ACTION _CalData:
// nOutputMode
// 0 : uses setpoint and setpoint type to control the valve.
// 1 : Does not use setpoint and setpoint type to operate the valve.
// 2 : Does not use setpoint and setpoint type to operate the valve.
// 3 : Holds valve in current position.
// 4 : Reset the controller.

GVL_IO.nIQPLUS_SetType 	:= GVL_DEVICE_NET_IQ_PLUS.nOutputSetType;
GVL_IO.nIQPLUS_Mode 	:= GVL_DEVICE_NET_IQ_PLUS.nOutputMode;
GVL_DEVICE_NET_IQ_PLUS.nOutputMode := GVL_COMMAND_FROM_UI.CMD_THROTTLE_OUTPUT_MODE;
GVL_IO.aMonitoring_PV[E_Morning_Index.E_Morning_TV_Position] := wByteValvePosition_PV/SetPointFactor;

(* Read from Device Value *)
// 2USINT to WORD
wByteCDG1_PV 		:= USINT_TO_WORD_jh(GVL_DEVICE_NET_IQ_PLUS.aInputPressurePV_CDG1);
wByteCDG2_PV 		:= USINT_TO_WORD_jh(GVL_DEVICE_NET_IQ_PLUS.aInputPressurePV_CDG2);
wByteValvePosition_PV:= USINT_TO_WORD_jh(GVL_DEVICE_NET_IQ_PLUS.aInputValvePosionPV);
wByteValvePosition_PV_Monitoring:=REAL_TO_WORD(wByteValvePosition_PV/SetPointFactor);
GVL_IO.aMonitoring_PV[12] := wByteValvePosition_PV_Monitoring;




wControlValue		:= GVL_IO.wIqPlus_CV;

//From IQ Plus
CDG1_RealValue :=wByteCDG1_PV/PressureFactor; 
GVL_IO.wIqPlus_CDG1_PV 	:= REAL_TO_WORD(wByteCDG1_PV/PressureFactor);
GVL_IO.wIqPlus_CDG2_PV:=GVL_IO.wIqPlus_CDG1_PV;

IF GVL_IO.wIqPlus_CDG1_PV > 800 OR GVL_IO.wIqPlus_CDG1_PV <=1 THEN
	GVL_IO.wIqPlus_CDG1_PV:=0;
	GVL_IO.wIqPlus_CDG2_PV:=0;
END_IF

CDG_1_Value_RealType:=wByteCDG1_PV/PressureFactor;


//nSetType //1:Pressure Conrol, 2:Position Control

IF GVL_DEVICE_NET_IQ_PLUS.nOutputMode = 0 AND nSetType = 1 THEN(*Pressure Mode*)
	wTypedControlValue := REAL_TO_WORD(wControlValue * SetPointFactor * 0.1); //Pressure Control
ELSIF GVL_DEVICE_NET_IQ_PLUS.nOutputMode = 0 AND nSetType = 2 THEN (*Position Mode*)
	wTypedControlValue := REAL_TO_WORD(wControlValue * SetPointFactor); // Position Control
END_IF

wOutputSVBytes 		:= WORD_TO_USINT_Bit(wTypedControlValue);
GVL_DEVICE_NET_IQ_PLUS.aOutputSVBytes[1] 	:= wOutputSVBytes.Lower;
GVL_DEVICE_NET_IQ_PLUS.aOutputSVBytes[2] 	:= wOutputSVBytes.Upper;

//Valve Status Initailize
IF GVL_DEVICE_NET_IQ_PLUS.nInputStatus <> nInputStatusOld THEN
	// Staus Initializing
	ingPressureControl := FALSE;
	ingPositionControl := FALSE;
	isValveOpen := FALSE;
	isValveNotInitialized := FALSE;	
	isValveClosed := FALSE;
	isValveFaultState := FALSE;
	ingValveInitializing := FALSE;
	ingHoldState := FALSE;
	isPressureControl:=FALSE;
	// Status Update	
	nInputStatusOld := GVL_DEVICE_NET_IQ_PLUS.nInputStatus;
END_IF

//Update Valve Status
CASE GVL_DEVICE_NET_IQ_PLUS.nInputStatus OF
	0 : ingPressureControl := TRUE; //Pressure Control Performing.
	1 : ingPositionControl := TRUE; //Position Control Performing.	
	2 : isValveOpen := TRUE; //Valve Open, Stopped, Not Controlling.
	3 : isValveNotInitialized := TRUE; //Valve not initialized power on or RESET Command.
	4 : isValveClosed := TRUE; //Valve Closed, Stopped, Not Controlling.
	5 : isValveFaultState := TRUE; //Has faulted during valve initialization or operation.
	6 : ingValveInitializing := TRUE; //Initailizing Process.
	7 :	isPressureControl:=TRUE;
	8 : ingHoldState := TRUE; //intermediate position, not at open or close and not controlling pressure.
END_CASE
END_ACTION

ACTION _DigitalInput:

(* Command *)

bPumpOn:= GVL_COMMAND_FROM_UI.CMD_VACUUM_PUMP_ON;
bPumpReset:=GVL_COMMAND_FROM_UI.CMD_VACUUM_PUMP_RESET;
(* Read from Power Distribution Pannel *)
bVacuumPumpCB		:= GVL_IO_GAS_CABINET.DI_02_VacuumPumpELCB;
bThrottleValveCP 	:= GVL_IO_GAS_CABINET.DI_02_T_VCP;

(* Read from Vacuum Pump *)
isPumpFault			:= GVL_IO_REACTOR_CABINET.DI_02_VacuumPumpFail;
isPumpWarning		:= GVL_IO_REACTOR_CABINET.DI_02_VacuumPumpWarning;
isPumpAlarm			:= GVL_IO_REACTOR_CABINET.DI_02_VacuumPumpAlarm;
isPumpRunning		:= GVL_IO_REACTOR_CABINET.DI_02_VacuumPumpFBRunning;
isFBRunning			:= GVL_IO_REACTOR_CABINET.DI_02_VacuumPumpRunning;


GVL_IO.isPumpRunning := GVL_IO_REACTOR_CABINET.DI_02_VacuumPumpFBRunning;
END_ACTION

ACTION _DigitalOutput:
//GVL_IO.aDigitalOutputIO[2].2 := bPumpOn; //Pump On
//GVL_IO.aDigitalOutputIO[2].3 := bPumpReset; // Pump Reset

GVL_IO_REACTOR_CABINET.DO_05_VacuumPumpStart_Stop := bPumpOn;
GVL_IO_REACTOR_CABINET.DO_05_VacuumPumpReset := bPumpReset;
END_ACTION

END_PROGRAM

// ---- POUs/P13_LineHeater.TcPOU
PROGRAM P13_LineHeater
VAR
	rTemperatureSV 		: ARRAY[1..8]OF REAL;
	bAutoTuneSV 		: ARRAY[1..8]OF BOOL;

	rTemperaturePV 		: ARRAY[1..8]OF REAL;
	isLineHeater_Run	: ARRAY[1..8]OF BOOL;
	isLineHeater_ATune	: ARRAY[1..8]OF BOOL;
	isLineHeater_Err	: ARRAY[1..8]OF BOOL;

	TimeOnDelay			: TON; //Time delay after Power ON of Thermal Bath
	TimeCycle			: TON;
	nComMode 			: INT; // //1 = PV Req, 2 = STATUS Req, 3 = SV Write, 4 = AutoTune On/Off
	nCount 				: INT;
	rTemperatureTV 		: ARRAY[1..8]OF REAL;
	bAutoTuneTV			: ARRAY[1..8]OF BOOL;

	//for sending variable
	TimeWaitSend		:TON;
	bSendingEnable 		: BOOL:=TRUE; // Check the Sending Stage
	bSetValueMode 		: BOOL;
	fbSend				: SendString;
	sSendString 		: STRING;
	bSendBusy			: BOOL;
	bSendingOK 			: BOOL; //v1
	eSendErrorID		: ComError_t;
	
	// for received variable
	TimeWaitReceive		:TON;
	fbReceive			: ReceiveString;
	sReceivedString		: STRING;
	bStringReceived		: BOOL;
	bReceiveBusy		: BOOL;
	bReceiveError		: BOOL;
	eReceiveErrorID		: ComError_t;
	bReceiveTimeout		: BOOL;
	bReceivedOK 		: BOOL;
	hStrReceivedST		: STRING;
	hStrReceivedPV		: STRING;
	
	nHeaterNumber 		: INT := 1;
	sHeaterNumber 		: STRING := '1';
	sReceivedHeaterNumber : STRING;
	nReceivedHeaterNumber : INT;
	sReceivedAffirmation : STRING;
	sReceivedData 		: STRING;
	nHeaterStrPositionPV : INT:= 11; //Received String Start Position
	nDecimal			:INT;
	nSendStrCounter		:INT := 1;
	bReset : BOOL;
	sTest : STRING;
	nStrPosition : INT;
	nHeaterNumberPV : INT;
	sTemperaturePV : STRING;
	(* Input *)
	bLineHeaterCB		: BOOL;
	bLineHeaterCP		: BYTE;
END_VAR

_DIgitalInput();

TimeOnDelay(IN:= GVL_IO_GAS_CABINET.DI_02_LineHeatersELCB, PT :=T#5S); //Time Delay after a Thermal Bath MC ON

IF TimeOnDelay.Q THEN
	TimeOnDelay(IN:=FALSE);
	FOR nHeaterNumber:= 1 TO 8 DO
		IF (rTemperatureTV[nHeaterNumber] <> rTemperatureSV[nHeaterNumber]) THEN
			// if SetValue are different to TargetValue, change Target vale to setvalue
			rTemperatureTV[nHeaterNumber] := rTemperatureSV[nHeaterNumber];
			
			_SendTemp();
		END_IF
	END_FOR
END_IF


rTemperaturePV[1] := GVL_Serial.LineHeater_data_1.LINE_HEATER_CH_1_PV_VALUE;
rTemperaturePV[2] := GVL_Serial.LineHeater_data_1.LINE_HEATER_CH_2_PV_VALUE;
rTemperaturePV[3] := GVL_Serial.LineHeater_data_1.LINE_HEATER_CH_3_PV_VALUE;
rTemperaturePV[4] := GVL_Serial.LineHeater_data_1.LINE_HEATER_CH_4_PV_VALUE;

rTemperaturePV[5] := GVL_Serial.LineHeater_data_2.LINE_HEATER_CH_1_PV_VALUE;
rTemperaturePV[6] := GVL_Serial.LineHeater_data_2.LINE_HEATER_CH_2_PV_VALUE;
rTemperaturePV[7] := GVL_Serial.LineHeater_data_2.LINE_HEATER_CH_3_PV_VALUE;
rTemperaturePV[8] := GVL_Serial.LineHeater_data_2.LINE_HEATER_CH_4_PV_VALUE;

GVL_IO.aLineHeater_rTemperaturePV := rTemperaturePV;

ACTION _DigitalInput:
bLineHeaterCB	:= GVL_IO_GAS_CABINET.DI_02_LineHeatersELCB;

bLineHeaterCP.0 	:= GVL_IO_GAS_CABINET.DI_03_LineHeater_1CP;
bLineHeaterCP.1 	:= GVL_IO_GAS_CABINET.DI_03_LineHeater_2CP;
bLineHeaterCP.2 	:= GVL_IO_GAS_CABINET.DI_03_LineHeater_3CP;
bLineHeaterCP.3 	:= GVL_IO_GAS_CABINET.DI_03_LineHeater_4CP;
bLineHeaterCP.4 	:= GVL_IO_GAS_CABINET.DI_03_LineHeater_5CP;
bLineHeaterCP.5 	:= GVL_IO_GAS_CABINET.DI_04_LineHeater_6CP;
bLineHeaterCP.6 	:= GVL_IO_GAS_CABINET.DI_04_LineHeater_7CP;
bLineHeaterCP.7 	:= GVL_IO_GAS_CABINET.DI_04_LineHeater_8CP;
END_ACTION

ACTION _SendTemp:
CASE nHeaterNumber OF
	1:
		GVL.fbLineHeater_Manager._SendModbusCommand(sendMessage:=F_Temp_Write_Set_Point(Module_Number:=1,CommandIndex:=16#0
																,Write_Value:=REAL_TO_WORD(rTemperatureSV[nHeaterNumber])));
	2:
		GVL.fbLineHeater_Manager._SendModbusCommand(sendMessage:=F_Temp_Write_Set_Point(Module_Number:=1,CommandIndex:=16#03E8
																,Write_Value:=REAL_TO_WORD(rTemperatureSV[nHeaterNumber])));
	3:
		GVL.fbLineHeater_Manager._SendModbusCommand(sendMessage:=F_Temp_Write_Set_Point(Module_Number:=1,CommandIndex:=16#07D0
																,Write_Value:=REAL_TO_WORD(rTemperatureSV[nHeaterNumber])));
	4:
		GVL.fbLineHeater_Manager._SendModbusCommand(sendMessage:=F_Temp_Write_Set_Point(Module_Number:=1,CommandIndex:=16#0BB8
																,Write_Value:=REAL_TO_WORD(rTemperatureSV[nHeaterNumber])));
																
	(*Change Module Number*)															
	5:
		GVL.fbLineHeater_Manager._SendModbusCommand(sendMessage:=F_Temp_Write_Set_Point(Module_Number:=2,CommandIndex:=16#0
																,Write_Value:=REAL_TO_WORD(rTemperatureSV[nHeaterNumber])));
	6:
		GVL.fbLineHeater_Manager._SendModbusCommand(sendMessage:=F_Temp_Write_Set_Point(Module_Number:=2,CommandIndex:=16#03E8
																,Write_Value:=REAL_TO_WORD(rTemperatureSV[nHeaterNumber])));
	7:
		GVL.fbLineHeater_Manager._SendModbusCommand(sendMessage:=F_Temp_Write_Set_Point(Module_Number:=2,CommandIndex:=16#07D0
																,Write_Value:=REAL_TO_WORD(rTemperatureSV[nHeaterNumber])));
	8:
		GVL.fbLineHeater_Manager._SendModbusCommand(sendMessage:=F_Temp_Write_Set_Point(Module_Number:=2,CommandIndex:=16#0BB8
																,Write_Value:=REAL_TO_WORD(rTemperatureSV[nHeaterNumber])));
END_CASE
END_ACTION

END_PROGRAM

// ---- POUs/P14_ThermalBath.TcPOU
PROGRAM P14_ThermalBath
VAR
	rTemperatureSV 		: ARRAY[1..6]OF REAL;

	(* Input from Device *)
	bTempDeviationAlarm	: ARRAY[1..6] OF BOOL;
	bCutOffAlarm		: ARRAY[1..6] OF BOOL;
	
	rTemperature_PV 		: ARRAY[1..6]OF REAL;
	isBath_Err 			: ARRAY[1..6]OF BOOL;
	isBath_TC_Broken 	: ARRAY[1..6]OF BOOL ; 

	//for send variable
	TimeOnDelay	: TON; //Time delay after Power ON of Thermal Bath
	TimeCycle			: TON;
	TimeWaitSend		: TON;
	TimeWaitReceive		: TON;
	bSendingEnable 		: BOOL:=TRUE; // Check the Sending Stage
	bSetValueMode 		: BOOL;
	rTemperatureTV 		: ARRAY[1..6]OF REAL;
	fbSend				: SendString;
	sSendString 		: STRING;
	bSendBusy			: BOOL;
	bSendingOK 			: BOOL;
	eSendErrorID		: ComError_t;

	// for received variable
	fbReceive			: ReceiveString;
	sReceivedString		: STRING;
	bStringReceived		: BOOL;
	bReceiveBusy		: BOOL;
	bReceiveError		: BOOL;
	eReceiveErrorID		: ComError_t;
	bReceiveTimeout		: BOOL;
	bReceivedOK 		: BOOL;
	
	nBathNumber 		: INT := 1;
	sBathNumber 		: STRING := '1';
	sReceivedBathNumber : STRING;
	nReceivedBathNumber : INT;
	sReceivedAffirmation : STRING;
	sReceivedData 		: STRING;
	
	(* Input *)
	bThermalBathCB		: BOOL;
	index				: INT;
END_VAR

// Call the send block every second to repeat the transmission.
// Also call the block as long as it is busy to finish a transmission.
//TB: Thermal Bath x 6EA
//Maker: SMC
//Model: HEBC002-WA10
//Temp Range: -15 ~60℃
//RS485: 9600, DataBit(8), Parity(None), StopBit(1)
//BCC Check X

(* Read from Power Distribution Pannel *)
_DigitalInput();

// make a sending string
TimeCycle(IN := TimeOnDelay.Q, PT := T#1S); //Cycle for Serial Communication
IF TimeCycle.Q = TRUE THEN
	TimeCycle(IN := FALSE);

	// Make a sending string Set value or Request value 
	IF bSendingEnable = TRUE THEN
		//Set sate
		bSendingEnable := FALSE;
		bReceivedOK := FALSE;
		bSetValueMode := FALSE;
		
		//Target value(Bath) Set value
		IF (rTemperatureTV[nBathNumber] <> rTemperatureSV[nBathNumber])  OR isBath_Err[nBathNumber] THEN
			
			rTemperatureTV[nBathNumber] := rTemperatureSV[nBathNumber];
			
			sSendString := Real_To_String_ThermalBath(rTemperatureTV[nBathNumber],nBathNumber); //Send a SetValue=10.0 '$0201WSV100100$03'
			bSetValueMode := TRUE;
		ELSE
			sBathNumber := INT_TO_STRING(nBathNumber);
			sSendString := INSERT('$020RPV1$03',sBathNumber,2); //Request a PV
			bSetValueMode := FALSE;
		END_IF
		
		// Send string	
		fbSend(	SendString:= sSendString,
			TXbuffer:= GVL_Serial.TxBufferTB,
			
			Busy=> bSendBusy,
			Error=> );
		IF fbSend.Error <> COMERROR_NOERROR THEN
			eSendErrorID := fbSend.Error;
			bSendingOK := FALSE;
		ELSE
			eSendErrorID := COMERROR_NOERROR;
			bSendingOK := TRUE;
		END_IF
		
	END_IF

	//	Receive string data:
	//	The block receives any data strings beginning with a STX ($02) and ending with an ETX ($03) character.
	TimeWaitReceive(IN := bSendingOK, PT := T#250MS); //Wait receiving data
	IF TimeWaitReceive.Q THEN
		TimeWaitReceive(IN:= FALSE);
		fbReceive(
			Prefix:= '$02',
			Suffix:= '$03',
			Timeout:= T#1S,
			ReceivedString:= sReceivedString,
			RXbuffer:= GVL_Serial.RxBufferTB,
			
			StringReceived=> bStringReceived,
			Busy=> bReceiveBusy,
			Error=> ,
			RxTimeout=> bReceiveTimeout );
			
		IF bReceiveTimeout THEN
			isBath_Err[nReceivedBathNumber] := TRUE;
			bReceiveTimeout := FALSE;
		END_IF
		
		IF fbReceive.Error <> COMERROR_NOERROR THEN
			eReceiveErrorID := fbReceive.Error;
		END_IF
		
		IF bStringReceived THEN
			bStringReceived :=FALSE;
			bReceivedOK := TRUE;
			bSendingEnable := TRUE;
			sReceivedBathNumber := MID(STR:=sReceivedString, len:=1, pos:=3); //ReceivedString : '$0201$06PV100250$03'
			nReceivedBathNumber := STRING_TO_INT(sReceivedBathNumber);
			sReceivedAffirmation := MID(STR:=sReceivedString, len:=1, pos:=4); //Affirmation
			
			IF bSetValueMode THEN //Write SV Mode
				IF sReceivedAffirmation = '$06' THEN //'$06' ReceivedString : '$0201$06$03'
					isBath_Err[nReceivedBathNumber] := FALSE;
				ELSE
					//isBath_Err[nReceivedBathNumber] := TRUE;
				END_IF
				bSetValueMode := FALSE;
			ELSE //Read PV Mode
				sReceivedData := MID(STR:=sReceivedString, len:=5, pos:=8); //ReceivedString : '$0201$06PV100250$03'
				IF sReceivedData = '' THEN
					//isBath_Err[nReceivedBathNumber] := TRUE;
				ELSIF sReceivedData = 'HHHHH' THEN
					rTemperature_PV[nReceivedBathNumber] := -99.0;
					isBath_TC_Broken[nReceivedBathNumber] := TRUE;
					isBath_Err[nReceivedBathNumber] := FALSE;
				ELSE
					rTemperature_PV[nReceivedBathNumber] := (STRING_TO_REAL(sReceivedData))/10;
					isBath_TC_Broken[nReceivedBathNumber] := FALSE;
					isBath_Err[nReceivedBathNumber] := FALSE;
				END_IF
			END_IF
			index := nReceivedBathNumber + 11;
			
			
		END_IF
	END_IF
	
	//Change the Next Bath
	nBathNumber := nBathNumber + 1;
	IF nBathNumber > 4 THEN
		nBathNumber := 1;
	END_IF
	bSendingEnable := TRUE;
END_IF

ACTION _DigitalInput:
//bThermalBathCB := GVL_IO.aDigitalInputIO[5].0;
bThermalBathCB := GVL_IO_GAS_CABINET.DI_02_ThermalBathsELCB;

(* Read from SMC Bath Device Value *)
//TimeOnDelay(IN:= P90_Interlock.bThermalBathMC, PT :=T#1S); //Time Delay after a Thermal Bath MC ON
TimeOnDelay(IN:= GVL_IO_GAS_CABINET.DI_02_ThermalBathsELCB, PT :=T#1S); //Time Delay after a Thermal Bath MC ON

bTempDeviationAlarm[1]	:= GVL_IO_GAS_CABINET.DI_05_ThermalBath_1DeviationAlarm;
bTempDeviationAlarm[2]	:= GVL_IO_GAS_CABINET.DI_05_ThermalBath_2DeviationAlarm;
bTempDeviationAlarm[3]	:= GVL_IO_GAS_CABINET.DI_06_ThermalBath_3DeviationAlarm;
bTempDeviationAlarm[4]	:= GVL_IO_GAS_CABINET.DI_06_ThermalBath_4DeviationAlarm;

bCutOffAlarm[1] := NOT(GVL_IO_GAS_CABINET.DI_05_ThermalBath_1CutOffAlarm); //Normally Contact
bCutOffAlarm[2] := NOT(GVL_IO_GAS_CABINET.DI_05_ThermalBath_2CutOffAlarm); 
bCutOffAlarm[3] := NOT(GVL_IO_GAS_CABINET.DI_06_ThermalBath_3CutOffAlarm); 
bCutOffAlarm[4] := NOT(GVL_IO_GAS_CABINET.DI_06_ThermalBath_4CutOffAlarm);
END_ACTION

END_PROGRAM

// ---- POUs/P15_RotationOperation.TcPOU
PROGRAM P15_RotationOperation
VAR
	rControlValue			: REAL; //rpm
	bStart_Stop				: BOOL := TRUE;
	bAlarmReset				: BOOL; //Motor Driver Alarm

	bRotationCP				: BOOL;
	nConvertedRotation_PV	: REAL; //PV 0~100 rpm

	rConvertedCV			:REAL;
	(* Motor Driver *)
	bBrake_Run				: BOOL;
	(* Rotation Operation Parameter*)
	wRotaion_PV				: WORD;
	isRotationFault			: BOOL; //Motor Driver
	calcRotation: REAL;
END_VAR

VAR CONSTANT
	KL4404MaxValueP		: REAL := 16383; //0~5V, 0~3000
	//Motor Max Rotation RPM 3000rpm, Gear Ratio 20, Belt Ratio 4.5
	ConversionFactor 	: REAL :=491.49;// 491.49 ; //13106 * 20 * 4.5 / 3000
END_VAR

// Oriental Motor Driver : BLHM230K-GFS, 0~4V

_DigitalInput();

calcRotation := (wRotaion_PV / ConversionFactor) * (5.0/3.0);


nConvertedRotation_PV := (calcRotation);

// Interface with other PRGs
GVL_IO.nRotation_Converted_PV := nConvertedRotation_PV;
rControlValue := GVL_IO.rRotation_ControlValue;

//Write to Motor Driver
rConvertedCV := rControlValue * ConversionFactor; // Convert from RPM to control value


IF GVL_io.aInterlockEnable[1].7 = TRUE THEN // UI 의 Auto Power ON 기능에 따라서 자동 On . oFF 사용 
	IF (GVL_IO.aController[E_aAnalogInputIO_Index.E_PV_susceptorRotation].input.targetValue > 0) OR (rConvertedCV > 0) THEN // Motor Driver RUN
		bBrake_Run := TRUE;
	ELSIF (GVL_IO.aController[E_aAnalogInputIO_Index.E_PV_susceptorRotation].input.targetValue = 0) AND (rConvertedCV = 0) THEN
		bBrake_Run := FALSE;
	END_IF
ELSE
	bBrake_Run:=FALSE;
END_IF

_DigitalOutput();

ACTION _DigitalInput:
(* Read from Power Distribution Pannel *)
bRotationCP := GVL_IO_GAS_CABINET.DI_02_RotationMotorCP;

//from Device Value
isRotationFault := NOT(GVL_IO_REACTOR_CABINET.DI_02_SusceptorRotationMotorFault);
wRotaion_PV := INT_TO_WORD(GVL_IO_REACTOR_CABINET.AI_08_R01SusceptorRotationPV);
END_ACTION

ACTION _DigitalOutput:
GVL_IO_REACTOR_CABINET.DO_05_SusceptorRotationFWD := bBrake_Run;
GVL_IO_REACTOR_CABINET.AO_09_R01_SusceptorRotationSV:=REAL_TO_INT(rConvertedCV);
END_ACTION

END_PROGRAM

// ---- POUs/P16_CoverOperation.TcPOU
PROGRAM P16_CoverOperation
VAR
// 	isCoverClosed 	: BOOL;

	bCoverCP	: BOOL;
	bLowerLimit	: BOOL;
	bUpperLimit	: BOOL;
	TimerUpLED 		: TON;
	TimerUpLED_X 	: TON;
	TimerDownLED 	: TON;
	TimerDownLED_X 	: TON;
	TimerDownDelayOff 	: TON;
	(* Input *)
	bUpSwitch	: BOOL;
	bDownSwitch 	: BOOL;
	bClamp_Lock_switch: BOOL;
	bClamp_Release_switch: BOOL;
	(* Output *)
	bUpLED 		: BOOL;
	bDownLED 	: BOOL;
	bOnUpRelay 	: BOOL;
	bOnDownRelay : BOOL;
	bOnClamp_Lock_Relay:BOOL;
	bOnClamp_Release_Relay:BOOL;		
	
	bClampLock: BOOL;
	bClampRelease: BOOL;
END_VAR

_DigitalInput();

TimerDownDelayOff(IN:=bLowerLimit, PT:=T#500MS);

//Cover Open 조건
//공정 중이지 않을것
//Dor Pressure down
//Clamp Releaae
//Susceptor down
//CDG 700 torr 이상
//모든 벨브 ff

// Cover Operation Condition
IF P90_Interlock.bReactorOpenEnable THEN
	(*Cover*)
	IF bClampRelease THEN
		bOnUpRelay := (bDownSwitch = FALSE AND bUpSwitch = TRUE AND bUpperLimit = FALSE );
		bOnDownRelay := (bDownSwitch = TRUE AND bUpSwitch = FALSE AND (bLowerLimit = FALSE OR TimerDownDelayOff.Q = FALSE ));
	ELSE
		bOnUpRelay:=FALSE;
		bOnDownRelay:=FALSE;
	END_IF
	(*clamp*)
	bOnClamp_Lock_Relay:=(bClamp_Lock_switch = TRUE AND bClamp_Release_switch = FALSE);
	bOnClamp_Release_Relay:=(bClamp_Lock_switch = FALSE AND bClamp_Release_switch = TRUE);
ELSE
	(*Cover*)
	bOnUpRelay:=FALSE;
	bOnDownRelay:=FALSE;
	(*clamp*)
	bOnClamp_Lock_Relay:=FALSE;
	bOnClamp_Release_Relay:=FALSE;
END_IF

//LED Blinking
TimerUpLED(IN:=(bOnUpRelay AND TimerUpLED_X.Q = FALSE), PT:=T#500MS);
TimerUpLED_X(IN:=TimerUpLED.Q, PT:=T#300MS);
bUpLED := (TimerUpLED.Q AND bOnUpRelay) OR bUpperLimit;

TimerDownLED(IN:=(bOnDownRelay AND TimerDownLED_X.Q = FALSE), PT:=T#500MS);
TimerDownLED_X(IN:=TimerDownLED.Q, PT:=T#300MS);
bDownLED := (TimerDownLED.Q AND bOnDownRelay) OR bLowerLimit;

_DigitalOutput();

ACTION _DigitalInput:
//(* Read from Device Value *)
//// Cover Operation Switch
//bUpSwitch 		:= GVL_IO.aDigitalInputIO[1].6;
//bDownSwitch 	:= GVL_IO.aDigitalInputIO[1].7;
//bUpperLimit 	:= GVL_IO.aDigitalInputIO[3].4;
//bLowerLimit 	:= GVL_IO.aDigitalInputIO[3].5;
//bCoverCP 		:=  GVL_IO.aDigitalInputIO[5].4;

bUpSwitch 		:=GVL_IO_REACTOR_CABINET.DI_01_ReactorDoorUpButton;
bDownSwitch 	:=GVL_IO_REACTOR_CABINET.DI_01_ReactorDoorDownButton;
bUpperLimit 	:=GVL_IO_REACTOR_CABINET.DI_02_ReactorDoorUpLimitSensor;
bLowerLimit 	:=GVL_IO_REACTOR_CABINET.DI_03_ReactorDoorDownLimitSensor;
bCoverCP 		:= GVL_IO_GAS_CABINET.DI_02_CoverLiftMotorCP;

bClampLock := GVL_IO_REACTOR_CABINET.DI_03_CylinderAutoSwitch_Closed;
bClampRelease :=GVL_IO_REACTOR_CABINET.DI_03_CylinderAutoSwitch_Opened;

bClamp_Lock_switch:=GVL_IO_REACTOR_CABINET.DI_01_ClampLock;
bClamp_Release_switch:=GVL_IO_REACTOR_CABINET.DI_01_ClampRelease;
END_ACTION

ACTION _DigitalOutput:
(* Write to Device Value *)
// Cover Operation Switch Lamp


//Status Output
GVL_IO.isCoverClosed := bLowerLimit;

GVL_IO_REACTOR_CABINET.DO_06_ReactorCoverUpButtonLamp := bUpLED;
GVL_IO_REACTOR_CABINET.DO_06_ReactorCoverDownButtonLamp := bDownLED;

GVL_IO_REACTOR_CABINET.DO_04_ReactorCoverUpRelay :=bOnUpRelay;
GVL_IO_REACTOR_CABINET.DO_04_ReactorCoverDownRelay :=bOnDownRelay;

GVL_IO_REACTOR_CABINET.DO_06_ClampLockButtonLamp := GVL_IO_REACTOR_CABINET.DI_03_CylinderAutoSwitch_Closed;
GVL_IO_REACTOR_CABINET.DO_06_ClampReleaseButtonLamp := GVL_IO_REACTOR_CABINET.DI_03_CylinderAutoSwitch_Opened;

GVL_IO_REACTOR_CABINET.DO_05_ClampLock := bOnClamp_Lock_Relay;
GVL_IO_REACTOR_CABINET.DO_05_ClampRelease := bOnClamp_Release_Relay;
END_ACTION

END_PROGRAM

// ---- POUs/P17_DOROperation.TcPOU
PROGRAM P17_DOROperation
VAR
	bDOROn				: BOOL; //UI Input Button
	bDOROff				: BOOL; //UI Input Button
	fTresholdPressure	: REAL;
	fTresholdCount		: REAL;
	bPressureEnable 	: BOOL;
	bCountEnable		: BOOL;

	isDOROnState		: BOOL := FALSE; //DOR ON State
	bError				: INT; //0: No Err, 1: Vacuum Fail, 2: Vacuum Release, 3: Try out
	nWaitCounter		: INT;

	(* Input *)
	bVacSwitch			: BOOL; //Push Switch
	bAtmSwitch			: BOOL; //Push Switch
	(* Pressure Transducer *)
	nPressurePV			: INT;
	rPressurePV_kPa		: REAL;
	(* Output *)
	bVacLED				: BOOL;
	bAtmLED				: BOOL;
	bV_DORVac			: BOOL; //V34 Valve
	bV_DORFill			: BOOL; //V35 Valve
	
	(* DOR Condition Operation Parameter *)
	rTrigSwitch			: R_TRIG;
	TimerOnLED			: TON;
	TimerVacSwitch		: TON;
	TimerAtmSwitch		: TON;
	TimerWaitCheck		: TON;
	TimerVacRealease	: TON;
	nCase				: INT := 0;
	nTresholdCount		: INT;
	nTryCount			: INT;
	bVacuumRealse		: BOOL;
	//Temperatur Variable
	bTest				: BOOL;
	nTest				: INT;
END_VAR

VAR CONSTANT
	KL3464MaxValueP		: REAL := 16383; //1 ~ 5VDC, 0 ~ 100kPa(1bar), PG35
	SlopeFactor			: REAL := 0.007617887; //100kPa/(16383-3256)
END_VAR

// Double O-Ring Vacuum Condition

_DigitalInput();

(* If Vacuum 'ON' Switch Press, Change DOR Vacuum State *)
//DOR Operation Signal generation

TimerVacSwitch(IN:=bVacSwitch OR bDOROn, PT:=T#100MS);
rTrigSwitch(CLK:=TimerVacSwitch.Q);

IF rTrigSwitch.Q AND GVL_IO.bDorOnEnable THEN
	nCase 		:= 1;
	nTryCount 	:= 1; //Try One more Vacuum 
END_IF

CASE nCase OF
	1: //Initialize
		isDOROnState := FALSE;
		bV_DORVac 	:= TRUE; //V34 Open
		bV_DORFill	:= FALSE; //V35 Close
		bAtmLED		:= FALSE;
		TimerWaitCheck(IN:=FALSE);	
		nCase := 10;
	10: //Wait and Vacuum Check
		(* Blink Switch LED *)
		TimerOnLED(IN:=TRUE, PT:=T#500MS);
		IF TimerOnLED.Q THEN
			TimerOnLED(IN:=FALSE);
			bVacLED := NOT(bVacLED);
		END_IF

		TimerWaitCheck(IN:=TRUE, PT:=T#5S);
		IF TimerWaitCheck.Q THEN
			IF rPressurePV_kPa > fTresholdPressure THEN
				bV_DORVac 		:= FALSE; //V34 Close
				isDOROnState 	:= TRUE;
				bVacLED 		:= TRUE; //Switch LED
				bError			:= 0;
				nCase 			:= 0;
			ELSIF nTryCount < nTresholdCount THEN
				TimerWaitCheck(IN:=FALSE);
				nTryCount 		:= nTryCount + 1;				
				nCase 			:= 1;
			ELSE
				bV_DORVac 		:= FALSE; //V34 Close
				isDOROnState 	:= FALSE;
				bVacLED			:= FALSE; //Switch LED
				bError			:= 1; // Vacuum Fail
				nCase			:= 0;
			END_IF
		END_IF
END_CASE

(* If Vacuum 'OFF' Switch Press, Change DOR Vent(Fill, Atm) State *)
//DOR Operation Signal generation
TimerAtmSwitch(IN:=bAtmSwitch OR bDOROff, PT:=T#100MS);
rTrigSwitch(CLK:=TimerAtmSwitch.Q);

IF rTrigSwitch.Q AND P90_Interlock.bDorOffEnable THEN
	nCase := 2;
END_IF

CASE nCase OF
	2:
		(* Blink Switch LED *)
		TimerOnLED(IN:=TRUE, PT:=T#500MS);
		IF TimerOnLED.Q THEN
			TimerOnLED(IN:=FALSE);
			bAtmLED := NOT(bAtmLED);
		END_IF
		
		TimerWaitCheck(IN:=TRUE, PT:=T#10S);
		nWaitCounter := TIME_TO_INT(TimerWaitCheck.ET/1000);
		IF TimerWaitCheck.Q THEN
			TimerWaitCheck(IN:=FALSE);
			bVacLED			:= FALSE;
			bV_DORVac 		:= FALSE; //V34 Close
			bV_DORFill		:= TRUE; //V35 Open
			nCase			:= 20;
		END_IF
	20:
		TimerWaitCheck(IN:=TRUE, PT:=T#5S);
		IF TimerWaitCheck.Q THEN
			bVacLED			:= FALSE;
			bV_DORFill		:= FALSE;
			isDOROnState 	:= FALSE;
			bAtmLED			:= TRUE;
			nCase			:= 0;
		END_IF
END_CASE

(* If Vacuum 'ON' State, Check the Vacuum range *)
IF isDOROnState AND rPressurePV_kPa < (fTresholdPressure - 20) AND nTryCount < 3 THEN
	bError := 2; // Vacuum release
	TimerVacRealease(IN:=TRUE, PT:=T#2S);
	
	(* Blink Vac Switch LED *)
	TimerOnLED(IN:=TRUE, PT:=T#500MS);
	IF TimerOnLED.Q THEN
		TimerOnLED(IN:=FALSE);
		bVacLED := NOT(bVacLED);
	END_IF

	IF TimerVacRealease.Q  THEN
		TimerVacRealease(IN:=FALSE);
		nTryCount 		:= nTryCount + 1;
		bV_DORVac 		:= FALSE;//Vacuum Valve OFF
		bVacLED := TRUE;
	ELSE
		bV_DORVac 		:= TRUE;//Vacuum Valve ON
	END_IF
	
ELSIF bError = 2 THEN
	bV_DORVac := FALSE;
	bError := 0;
	
ELSIF nTryCount >= 3 THEN
	bV_DORVac := FALSE;
	bError := 3; //Vacuum Released
END_IF

//알람 리셋
IF GVL_IO.aInterlockEnable[1].0 OR GVL_IO.aInterlockEnable[1].1 THEN
	bError := 0;
END_IF

_DigitalOutput();

ACTION _DigitalInput:
(* Read from Device Value *)
// DOR Operation Switch
bVacSwitch 			:= GVL_IO_REACTOR_CABINET.DI_01_DORVACButton; //Switch Input
bAtmSwitch 			:= GVL_IO_REACTOR_CABINET.DI_01_DORATMButton; //Switch Input
nPressurePV 		:= GVL_IO_REACTOR_CABINET.AI_07_S05_DORPressurePV;
rPressurePV_kPa 	:= F_GetDorPressure(nPressurePV);

fTresholdPressure 	:= GVL_IO.aInterlockSet[11]; // Dor Pressure Limit
fTresholdCount 		:= GVL_IO.aInterlockSet[12]; // Dor Retry Count

bPressureEnable 	:= GVL_IO.aInterlockEnable[1].5; // Dor Pressure Limit
bCountEnable 		:= GVL_IO.aInterlockEnable[1].6; // Dor Retry Count
nTresholdCount 		:= REAL_TO_INT(fTresholdCount); //Try One more Vacuum
END_ACTION

ACTION _DigitalOutput:
(* Write to Device Value *)
// Cover Operation Switch Lamp

//GVL_IO_VALVE.DO_00_V22DORVaccumON :=GVL_IO.aOutputSolValve[2].5;
//GVL_IO_VALVE.DO_00_V23DORFilling :=GVL_IO.aOutputSolValve[2].6;

GVL_IO.aOutputSolValve.21:= bV_DORVac; //V34
GVL_IO.aOutputSolValve.22:= bV_DORFill; //V35

GVL_IO.aInputState[4].10 :=bV_DORVac;

GVL_IO_REACTOR_CABINET.DO_05_DORVACButtonLamp := bVacLED;
GVL_IO_REACTOR_CABINET.DO_06_DORATMButtonLamp := bAtmLED;

GVL_IO.nDorOperationError := bError;
//jhkang isDOROnState 뭐냐 
GVL_IO.bDorState := isDOROnState;
END_ACTION

END_PROGRAM

// ---- POUs/P30_ManualControl.TcPOU
Program P30_ManualControl
VAR
	analogDeviceRampControl : FB_AnalogDeviceRampControl;
END_VAR

analogDeviceRampControl();

END_PROGRAM

// ---- POUs/FB_AnalogDeviceRampControl.TcPOU
FUNCTION_BLOCK FB_AnalogDeviceRampControl
VAR
	i : INT;
END_VAR

FOR i:=1 TO E_aAnalogInputIO_Index.E_PV_EPC_04 DO
	GVL_IO.aAnalogOutputIO[i] := LREAL_TO_INT(GVL_IO.aController[i].rControlValue / GVL_CONSTANT.AnalogControllerOutputVoltage * GVL_CONSTANT.EL3064MaxValueH); //Write to Device
	GVL_IO.aController[i]();
END_FOR


//jhkang aController 의 Input은 언제 들어감?
//Temp Controller
GVL_IO.wE3508_CV := LREAL_TO_WORD(GVL_IO.aController[E_aAnalogInputIO_Index.E_PV_Susceptor_Temp].rControlValue * 10 )  ; //Write to Temperature Controller
GVL_IO.aController[E_aAnalogInputIO_Index.E_PV_Susceptor_Temp]();

//Temp Pressure Controller				
GVL_IO.wIqPlus_CV := LREAL_TO_WORD(GVL_IO.aController[E_aAnalogInputIO_Index.E_PV_Reactor_Pressure].rControlValue); //Write to Pressure Controller
GVL_IO.aController[E_aAnalogInputIO_Index.E_PV_Reactor_Pressure]();

//Rotation Controller		
GVL_IO.rRotation_ControlValue := LREAL_TO_REAL(GVL_IO.aController[E_aAnalogInputIO_Index.E_PV_susceptorRotation].rControlValue); //Write to Rotation Controller (rpm)
GVL_IO.aController[E_aAnalogInputIO_Index.E_PV_susceptorRotation]();

END_FUNCTION_BLOCK

// ---- POUs/P50_RecipeControl.TcPOU
PROGRAM P50_RecipeControl
VAR
	nRcpIndex		: INT;
	eRecipeRun		: E_RecipeRun ; //레시피 상태
	fbAnalogDeviceRampControl : FB_AnalogDeviceRampControl;
	fbRecipeAnalogInputControlSequencer: FB_RecipeAnalogControlInputSequencer;
	fbOnlyPVUpdate: FB_OnlyPVUpdate;
	fbValveControl: FB_ValveControl;
	
	Pause_TON		: TON;
	Ramp_TON		: FB_TON_Pausable;
	Hold_TON		: FB_TON_Pausable;
	
	loopCount		: ARRAY[1..100] OF INT;
	i				: INT;
END_VAR
VAR CONSTANT
	Pause_MAX		: TIME := T#1800S;
END_VAR

CASE RCP.cmd_RcpOperation OF
	0: //Init State
 		f_ResetTimersAndRCPTimes(fbPause_TON := Pause_TON, fbRamp_TON := Ramp_TON, fbHold_TON := Hold_TON);
		
		FOR i:=1 TO Rcp.iRcpTotalStep DO
			loopCount[i] := Rcp.aRecipe[i].iRecipe[5];
		END_FOR
		
		nRcpIndex := 0;
		Rcp.userState := 0;
		eRecipeRun := E_RecipeRun.Initial;
		GVL_IO.nCaseSignalTower := 5; // White - Idle

	10: //RUN
		IF nRcpIndex = 0 THEN
			nRcpIndex := 1;
		END_IF
		fbAnalogDeviceRampControl();
						
		// CASE 문을 이용한 상태 머신 구현
		CASE eRecipeRun OF
			E_RecipeRun.Initial:
				f_ResetTimersAndRCPTimes(fbPause_TON := Pause_TON, fbRamp_TON := Ramp_TON, fbHold_TON := Hold_TON);
				fbRecipeAnalogInputControlSequencer(rRecipe := RCP.aRecipe[nRcpIndex].rRecipe, rampTime:= TO_UINT(RCP.aRecipe[nRcpIndex].iRecipe[2]));
				fbValveControl(valveSetting:= RCP.aRecipe[nRcpIndex].dRecipe);
				Rcp.userState := 10;// Recipe Running
				GVL_IO.nCaseSignalTower := 3;
				eRecipeRun := E_RecipeRun.Ramp;
				
			E_RecipeRun.Ramp: // Ramp 수행
				Ramp_TON(IN:=TRUE, PT:= RCP.aRecipe[nRcpIndex].iRecipe[2] * T#1S, ET=>RCP.RecipeRunET.ET);
				RCP.RecipeRunET.Mode := E_RecipeRunETMode.Ramp;
				IF Ramp_TON.Q THEN
					Ramp_TON(IN:=FALSE);
					eRecipeRun := E_RecipeRun.CheckHoldTemp;
				END_IF				
				
			E_RecipeRun.CheckHoldTemp: //Hold Temp 확인
				IF RCP.aRecipe[nRcpIndex].cTemp = 0.0 THEN
					Hold_TON(IN:=TRUE, PT:= RCP.aRecipe[nRcpIndex].iRecipe[3] * T#1S, ET=>RCP.RecipeRunET.ET);
					RCP.RecipeRunET.Mode := E_RecipeRunETMode.Hold;
					IF Hold_TON.Q THEN
						Hold_TON(IN:=FALSE);
						eRecipeRun := E_RecipeRun.End; // 레시피 첫 Column 실행
					END_IF
				ELSIF GVL_IO.aController_PV[E_aAnalogInputIO_Index.E_PV_Susceptor_Temp] < RCP.aRecipe[nRcpIndex].cTemp THEN //서셉터 온도가 Wait 온도보다 낮을 때
					Hold_TON(IN:=FALSE);
					eRecipeRun := E_RecipeRun.End; // 레시피 첫 Column 실행
				ELSE // 서셉터 온도가 Wait 온도보다 높을 때
					;// 떨어질 때까지 기다림
				END_IF
				
			E_RecipeRun.End: // 다음 Step 이동 (루프 마지막 단계일 경우, 다음 Step 이동 또는 루프 처음단계로 점프)
				loopCount[nRcpIndex] := loopCount[nRcpIndex] - 1;
				nRcpIndex := nRcpIndex + 1 - (RCP.aRecipe[nRcpIndex].iRecipe[4]) * MIN(loopCount[nRcpIndex], 1);
				IF nRcpIndex > Rcp.iRcpTotalStep THEN
					RCP.cmd_RcpOperation := 50;
				END_IF
				eRecipeRun := E_RecipeRun.Initial;
		END_CASE
		
	20: //PAUSE
		CASE eRecipeRun OF
			E_RecipeRun.Ramp:
				Ramp_TON(PAUSE:=TRUE);		
			E_RecipeRun.CheckHoldTemp:
				Hold_TON(PAUSE:=TRUE);
		END_CASE
		fbOnlyPVUpdate();
		
		Pause_TON(IN:=TRUE, PT:= Pause_MAX, ET=>RCP.Pause_ET); //최대 홀드 시간이 지나면 다음 스텝으로 넘거감
		IF Pause_TON.Q THEN
			Pause_TON(IN:=FALSE);
			eRecipeRun := E_RecipeRun.End; // 레시피 첫 Column 실행
		END_IF

		Rcp.userState := 20;
		GVL_IO.nCaseSignalTower := 5;
		
	30: //RESTART
		Pause_TON(IN:=FALSE);
		CASE eRecipeRun OF
			E_RecipeRun.Ramp:
				Ramp_TON(PAUSE:=FALSE);
			
			E_RecipeRun.CheckHoldTemp:
				Hold_TON(PAUSE:=FALSE);
		END_CASE

		RCP.Pause_ET := T#0S;
		Rcp.userState := 10;
		RCP.cmd_RcpOperation := 10;	
		GVL_IO.nCaseSignalTower := 3;
		
	40: //STOP
		f_ResetTimersAndRCPTimes(fbPause_TON := Pause_TON, fbRamp_TON := Ramp_TON, fbHold_TON := Hold_TON);
		F_StopAnalogRamping_ForRecipe();
		Rcp.userState := 40;
		GVL_IO.nCaseSignalTower := 5;
		
	50: //END
		f_ResetTimersAndRCPTimes(fbPause_TON := Pause_TON, fbRamp_TON := Ramp_TON, fbHold_TON := Hold_TON);
		Rcp.userState := 50;
		fbAnalogDeviceRampControl();
		GVL_IO.nCaseSignalTower := 5;
		
	60: //SKIP
		IF E_RecipeRun.Ramp <= eRecipeRun  AND  eRecipeRun <= E_RecipeRun.CheckHoldTemp THEN
			eRecipeRun := E_RecipeRun.End;
		END_IF
		Rcp.cmd_RcpOperation := 10;
		RCP.Pause_ET := T#0S;
END_CASE
RCP.iRcpStepN := nRcpIndex;

END_PROGRAM

// ---- POUs/FB_RecipeAnalogControlInputSequencer.TcPOU
FUNCTION_BLOCK FB_RecipeAnalogControlInputSequencer
VAR_INPUT
	rampTime: UINT;
END_VAR
VAR_IN_OUT
	rRecipe: ARRAY[1..(GVL_CONSTANT.NumAnalogController)] OF REAL;
END_VAR
VAR
	i: UINT;
END_VAR

FOR i:= 1 TO GVL_CONSTANT.NumAnalogController DO
	GVL_IO.aController[i].input.restart := TRUE;
	GVL_IO.aController[i].input.rampTime := rampTime; 
	GVL_IO.aController[i].input.targetValue := rRecipe[i];
END_FOR

END_FUNCTION_BLOCK

// ---- POUs/FB_OnlyPVUpdate.TcPOU
FUNCTION_BLOCK FB_OnlyPVUpdate
VAR_INPUT
END_VAR
VAR_OUTPUT
END_VAR
VAR
	i: INT;
END_VAR

FOR i:=1 TO E_aAnalogInputIO_Index.E_PV_EPC_04 DO
	IF 0.0 < GVL_IO.aMaxValueController[i]  THEN		
		GVL_IO.aController_PV[i] := (GVL_IO.aAnalogInputIO[i] / GVL_CONSTANT.EL3064MaxValueH) * GVL_IO.aMaxValueController[i];
	END_IF
END_FOR

GVL_IO.aController_PV[E_aAnalogInputIO_Index.E_PV_Susceptor_Temp] := WORD_TO_REAL(GVL_IO.wE3508_PV);
GVL_IO.aController_PV[E_aAnalogInputIO_Index.E_PV_Reactor_Pressure] := WORD_TO_REAL(GVL_IO.wIqPlus_CDG2_PV);
GVL_IO.aController_PV[E_aAnalogInputIO_Index.E_PV_susceptorRotation] := GVL_IO.nRotation_Converted_PV;

END_FUNCTION_BLOCK

// ---- POUs/FB_ValveControl.TcPOU
FUNCTION_BLOCK FB_ValveControl
VAR_INPUT
	valveSetting: DWORD; 
END_VAR

(* Solenoid Valve Mapping *)
GVL_IO.aOutputSolValve.0 := valveSetting.0; //V01 B/G N2 In
GVL_IO.aOutputSolValve.1 := valveSetting.1;
GVL_IO.aOutputSolValve.2 := valveSetting.2;
GVL_IO.aOutputSolValve.3 := valveSetting.3;
GVL_IO.aOutputSolValve.4 := valveSetting.4;
GVL_IO.aOutputSolValve.5 := valveSetting.5;
GVL_IO.aOutputSolValve.6 := valveSetting.6;
GVL_IO.aOutputSolValve.7 := valveSetting.7;

GVL_IO.aOutputSolValve.8 := valveSetting.8;
GVL_IO.aOutputSolValve.9 := valveSetting.9;
GVL_IO.aOutputSolValve.10 := valveSetting.10;
GVL_IO.aOutputSolValve.11 := valveSetting.11;
GVL_IO.aOutputSolValve.12 := valveSetting.12;
GVL_IO.aOutputSolValve.13 := valveSetting.13;
GVL_IO.aOutputSolValve.14 := valveSetting.14;
GVL_IO.aOutputSolValve.15 := valveSetting.15;

GVL_IO.aOutputSolValve.16 := valveSetting.16; 
GVL_IO.aOutputSolValve.17 := valveSetting.17;
GVL_IO.aOutputSolValve.18 := valveSetting.18;
GVL_IO.aOutputSolValve.19 := valveSetting.19;
GVL_IO.aOutputSolValve.20 := valveSetting.20;

END_FUNCTION_BLOCK

// ---- POUs/F_StopAnalogRamping_ForRecipe.TcPOU
FUNCTION F_StopAnalogRamping_ForRecipe
VAR
	i: UINT;
END_VAR

FOR i:= 1 TO GVL_CONSTANT.NumAnalogController DO
	GVL_IO.aController[i].input.restart := TRUE;
	GVL_IO.aController[i].input.rampTime := 1; 
	GVL_IO.aController[i].input.targetValue := LREAL_TO_REAL(GVL_IO.aController[i].rControlValue);
END_FOR

END_FUNCTION

// ---- POUs/P70_Interface.TcPOU
PROGRAM P70_Interface
VAR
END_VAR

//(* UI Right Dashboard Variable*)
//GVL_IO.aInputState[1].0 	:= GVL_IO.aDigitalInputIO[1].0; //Maintenance Key

//// GVL_IO.aInputState[1].1		:= P92_Maintenance.bReactorCabinetLamp; //Reactor Cabinet Lamp
//// GVL_IO.aInputState[1].2		:= P92_Maintenance.bGasCabinetLamp; // Gas Cabinet Lamp
//// GVL_IO.aInputState[1].3		:= P92_Maintenance.bPowerDistributeLamp; // Power Cabinet Lamp
//GVL_IO.aInputState[1].1		:= GVL_IO.aDigitalOutputIO[2].5; //Reactor Cabinet Lamp
//GVL_IO.aInputState[1].2		:= GVL_IO.aDigitalOutputIO[2].6; // Gas Cabinet Lamp
//GVL_IO.aInputState[1].3		:= GVL_IO.aDigitalOutputIO[2].7; // Power Cabinet Lamp

//GVL_IO.aInputState[1].4 	:= GVL_IO.aDigitalInputIO[2].0; //CDA Alarm Switch
//GVL_IO.aInputState[1].5		:= GVL_IO.aDigitalInputIO[2].1; //Water Flow Sensor

//// GVL_IO.aInputState[1].6 	:= P11_E3508.isHeaterReady; //Induction Heater
//// GVL_IO.aInputState[1].7 	:= P11_E3508.isHeaterRun; //Induction Heater
//// GVL_IO.aInputState[1].8 	:= P11_E3508.isHeaterFault; //Induction Heater
//GVL_IO.aInputState[1].6 	:= GVL_IO.aDigitalInputIO[2].2; //Induction Heater
//GVL_IO.aInputState[1].7 	:= GVL_IO.aDigitalInputIO[2].3; //Induction Heater
//GVL_IO.aInputState[1].8 	:= GVL_IO.aDigitalInputIO[2].4; //Induction Heater

//// GVL_IO.aInputState[1].9	:= P15_RotationOperation.bStart_Stop; //Susceptor Rotation Motor
//// GVL_IO.aInputState[1].10	:= P15_RotationOperation.bBrake_Run; //Susceptor Rotation Motor
//// GVL_IO.aInputState[1].11	:= P15_RotationOperation.isRotationFault; //Susceptor Rotation Motor
//GVL_IO.aInputState[1].9		:= GVL_IO.aDigitalOutputIO[3].4; //Susceptor Rotation Motor
//GVL_IO.aInputState[1].10	:= GVL_IO.aDigitalOutputIO[3].5; //Susceptor Rotation Motor

//// GVL_IO.aInputState[1].12 	:= P12_IQ_PLUS.isPumpWarning; //Vacuum Pump
//// GVL_IO.aInputState[1].13 	:= P12_IQ_PLUS.isPumpRunning; //Vacuum Pump
//// GVL_IO.aInputState[1].14 	:= P12_IQ_PLUS.isPumpFault; //Vacuum Pump
//GVL_IO.aInputState[1].12 	:= GVL_IO.aDigitalInputIO[3].0; //Vacuum Pump
//GVL_IO.aInputState[1].13 	:= GVL_IO.aDigitalInputIO[3].3; //Vacuum Pump
//GVL_IO.aInputState[1].14 	:= GVL_IO.aDigitalInputIO[2].7; //Vacuum Pump

//// GVL_IO.aInputState[1].15	:= P92_Maintenance.bReactorCabientMagnet; //Door Sensor
//GVL_IO.aInputState[1].15	:= GVL_IO.aDigitalInputIO[3].6; //Door Sensor

//// GVL_IO.aInputState[2].0		:= P92_Maintenance.bGasCabinetMagnet; //Door Sensor
//// GVL_IO.aInputState[2].1		:= P92_Maintenance.bPowerDistributeMagnet; //Door Sensor
//GVL_IO.aInputState[2].0		:= GVL_IO.aDigitalInputIO[3].7; //Door Sensor
//GVL_IO.aInputState[2].1		:= GVL_IO.aDigitalInputIO[4].0; //Door Sensor

//// GVL_IO.aInputState[2].2		:= P90_Interlock.bPowerResetSwitch; //Power Reset Switch
//GVL_IO.aInputState[2].2		:= GVL_IO.aDigitalInputIO[1].1; //Power Reset Switch

//// GVL_IO.aInputState[2].3		:= P16_CoverOperation.bUpperLimit; //Cover Upper Limit Sensor
//// GVL_IO.aInputState[2].4		:= P16_CoverOperation.bLowerLimit; //Cover Upper Limit Sensor
//GVL_IO.aInputState[2].3		:= GVL_IO.aDigitalInputIO[3].4; //Cover Upper Limit Sensor
//GVL_IO.aInputState[2].4		:= GVL_IO.aDigitalInputIO[3].5; //Cover Upper Limit Sensor

//// GVL_IO.aInputState[2].5		:= P92_Maintenance.bSMPS24V480WFault; //SMPS
//// GVL_IO.aInputState[2].6		:= P92_Maintenance.bSMPS24V72WFault;
//// GVL_IO.aInputState[2].7		:= P92_Maintenance.bSMPS15VPlusFault;
//// GVL_IO.aInputState[2].8		:= P92_Maintenance.bSMPS15VMinusFault;
//GVL_IO.aInputState[2].5		:= NOT(GVL_IO.aDigitalInputIO[4].3); //SMPS
//GVL_IO.aInputState[2].6		:= NOT(GVL_IO.aDigitalInputIO[4].4); 
//GVL_IO.aInputState[2].7		:= NOT(GVL_IO.aDigitalInputIO[4].5); 
//GVL_IO.aInputState[2].8		:= NOT(GVL_IO.aDigitalInputIO[4].6); 

//// GVL_IO.aInputState[2].9		:= P11_E3508.bInductionHeaterCB;
//GVL_IO.aInputState[2].9		:= GVL_IO.aDigitalInputIO[4].7;
//// GVL_IO.aInputState[2].10	:= P14_ThermalBath.bThermalBathCB;
//GVL_IO.aInputState[2].10	:= GVL_IO.aDigitalInputIO[5].0;
//// GVL_IO.aInputState[2].11	:= P12_IQ_PLUS.bVacuumPumpCB;
//GVL_IO.aInputState[2].11	:= GVL_IO.aDigitalInputIO[5].1;
//// GVL_IO.aInputState[2].12	:= P13_LineHeater.bLineHeaterCB;
//GVL_IO.aInputState[2].12	:= GVL_IO.aDigitalInputIO[5].2;
//// GVL_IO.aInputState[2].13	:= P15_RotationOperation.bRotationCP;
//GVL_IO.aInputState[2].13	:= GVL_IO.aDigitalInputIO[5].3;
//// GVL_IO.aInputState[2].14	:= P16_CoverOperation.bCoverCP;
//GVL_IO.aInputState[2].14	:= GVL_IO.aDigitalInputIO[5].4;
//// GVL_IO.aInputState[2].15	:= P12_IQ_PLUS.bThrottleValveCP;
//GVL_IO.aInputState[2].15	:= GVL_IO.aDigitalInputIO[5].5;

//GVL_IO.aInputState[3].0		:= GVL_IO.aDigitalInputIO[5].6;
//GVL_IO.aInputState[3].1		:= GVL_IO.aDigitalInputIO[5].7;

//GVL_IO.aInputState[3].2		:= GVL_IO.aDigitalInputIO[6].0; //Line Heater #1
//GVL_IO.aInputState[3].3		:= GVL_IO.aDigitalInputIO[6].1;
//GVL_IO.aInputState[3].4		:= GVL_IO.aDigitalInputIO[6].2;
//GVL_IO.aInputState[3].5		:= GVL_IO.aDigitalInputIO[6].3;
//GVL_IO.aInputState[3].6		:= GVL_IO.aDigitalInputIO[6].4;
//GVL_IO.aInputState[3].7		:= GVL_IO.aDigitalInputIO[6].5;
//GVL_IO.aInputState[3].8		:= GVL_IO.aDigitalInputIO[6].6;
//GVL_IO.aInputState[3].9		:= GVL_IO.aDigitalInputIO[6].7; //Line Heater #8
//GVL_IO.aInputState[3].10	:= GVL_IO.aDigitalInputIO[8].0; //Thermal Bath Temp. Deviation Alarm #1
//GVL_IO.aInputState[3].11	:= GVL_IO.aDigitalInputIO[8].2;
//GVL_IO.aInputState[3].12	:= GVL_IO.aDigitalInputIO[8].4;
//GVL_IO.aInputState[3].13	:= GVL_IO.aDigitalInputIO[8].6;
//GVL_IO.aInputState[3].14	:= GVL_IO.aDigitalInputIO[9].0;
//GVL_IO.aInputState[3].15	:= GVL_IO.aDigitalInputIO[9].2; //Thermal Bath Temp. Deviation Alarm #6

//GVL_IO.aInputState[4].0		:= GVL_IO.aDigitalOutputIO[1].0; // RED - Alarm
//GVL_IO.aInputState[4].1		:= GVL_IO.aDigitalOutputIO[1].1; // YELLOW - Waring
//GVL_IO.aInputState[4].2		:= GVL_IO.aDigitalOutputIO[1].2; // GREEN - Running
//GVL_IO.aInputState[4].3		:= GVL_IO.aDigitalOutputIO[1].3; // BLUE - Maintenance
//GVL_IO.aInputState[4].4		:= GVL_IO.aDigitalOutputIO[1].4; // WHITE - Idle
//GVL_IO.aInputState[4].5		:= GVL_IO.aDigitalOutputIO[1].5; // BUZZER - Alarm

//GVL_IO.aInputState[4].6		:= GVL_IO.aDigitalOutputIO[4].0; // DOR Vacuum State

//// GVL_IO.aInputState[4].7		:= P11_E3508.nInputAlarmBytes.7; // Temp Conroller Alarm State
//// GVL_IO.aInputState[4].8		:= P11_E3508.nInputManAutoBytes.7; // Temp Controller Mode State

//// P90_Interlock.bInductionHeaterMC := GVL_IO.aOutputCmd[1].0;
//// P90_Interlock.bThermalBathMC := GVL_IO.aOutputCmd[1].1;
//// P90_Interlock.bVacuumPumpMC := GVL_IO.aOutputCmd[1].2;
//// P90_Interlock.bLineHeaterMC := GVL_IO.aOutputCmd[1].3;

//// P11_E3508.bOutputManAuto := GVL_IO.aOutputCmd[1].11; //Temp Controller Mode Command
//// P12_IQ_PLUS.bPumpOn := GVL_IO.aOutputCmd[1].6

END_PROGRAM

// ---- POUs/P91_Monitoring.TcPOU
PROGRAM P91_Monitoring
VAR
	TimeCycle			: TON;
	i 					: INT;
	idx					: INT;
	
	(*Utility Input*)
	bUtilityFault		: BYTE;	
	JhValue_DOR: REAL;
	JhValue_EXHAUST: REAL;
END_VAR

//jhkang

(* Read from Utility Device*)

//jhkang butilityFault 는 어떤 것인가?
bUtilityFault.0		:= GVL_IO_GAS_CABINET.DI_05_ExternalH2GasCabinetFault;
bUtilityFault.1		:= GVL_IO_GAS_CABINET.DI_05_ExternalH2SGasCabinetFault;
bUtilityFault.2		:= GVL_IO_GAS_CABINET.DI_05_ExternalH2SeGasCabinetFault;
bUtilityFault.3		:= GVL_IO_GAS_CABINET.DI_05_ExternalUserInputAlarm;

TimeCycle(IN:=TRUE, PT:=T#100MS); // 100MS Refresh Reading Time
IF TimeCycle.Q THEN
	TimeCycle(IN:=FALSE);
	_DOR_EXHAUST();
	// Reactor Ultimate Pressure Gauge
	GVL_IO.aMonitoring_PV[1] := GVL_IO.aAnalogInputIO[E_aAnalogInputIO_Index.E_PV_Ultimate_Pressure] / GVL_CONSTANT.EL3064MaxValue * 10; //Ultimate Pressure 10Torr, 0~10V, Cal. x10
	GVL_IO.aMonitoring_PV[2] := JhValue_EXHAUST;
	GVL_IO.aMonitoring_PV[3] := JhValue_DOR;
	GVL_IO.aMonitoring_PV[4] := GVL_IO.aAnalogInputIO[E_aAnalogInputIO_Index.E_PV_GAS_Pressure_N2] / GVL_CONSTANT.EL3064MaxValue * 10; //N2 Cal. 6.89 bar  
	GVL_IO.aMonitoring_PV[5] := GVL_IO.aAnalogInputIO[E_aAnalogInputIO_Index.E_PV_GAS_Pressure_H2] / GVL_CONSTANT.EL3064MaxValue * 10; //H2 Cal. 6.89 bar
	GVL_IO.aMonitoring_PV[6] := GVL_IO.aAnalogInputIO[E_aAnalogInputIO_Index.E_PV_GAS_Pressure_H2S] / GVL_CONSTANT.EL3064MaxValue * 10; //NH3 Cal. 6.89 bar
	GVL_IO.aMonitoring_PV[7] := GVL_IO.aAnalogInputIO[E_aAnalogInputIO_Index.E_PV_GAS_Pressure_H2Se] / GVL_CONSTANT.EL3064MaxValue * 10; // Cal. 6.89 bar
	GVL_IO.aMonitoring_PV[8] := GVL_IO.aAnalogInputIO[E_aAnalogInputIO_Index.E_PV_CoolingWafer_SH] * 0.1; //  // PT100, Shower Head, Cal. 0.1
	GVL_IO.aMonitoring_PV[9] := GVL_IO.aAnalogInputIO2[1] / GVL_CONSTANT.EL3102MAxValue * 10;
	GVL_IO.aMonitoring_PV[10] := GVL_IO.aAnalogInputIO2[2] / GVL_CONSTANT.EL3102MAxValue * 10 ; 
	GVL_IO.aMonitoring_PV[11] := WORD_TO_REAL(P11_E3508.wE3508_PowerRate)*0.1; //divided to 10 PowerRate
	GVL_IO.aMonitoring_PV[12] := P12_IQ_PLUS.wByteValvePosition_PV_Monitoring;
	GVL_IO.aMonitoring_PV[13] := P14_ThermalBath.rTemperature_PV[1];
	GVL_IO.aMonitoring_PV[14] := P14_ThermalBath.rTemperature_PV[2];
	GVL_IO.aMonitoring_PV[15] := P14_ThermalBath.rTemperature_PV[3];
	GVL_IO.aMonitoring_PV[16] := P14_ThermalBath.rTemperature_PV[4];
END_IF

ACTION _DOR_EXHAUST:
GVL_SEQUENCE.FB_DOR_PRESSURE_AVG(newValue:=F_GetDorPressure(GVL_IO.aAnalogInputIO[E_aAnalogInputIO_Index.E_PV_DOR_PRESSURE]),Output=>JhValue_DOR);
GVL_SEQUENCE.FB_EXHAUST_AVG(newValue:=F_GetDorPressure(GVL_IO.aAnalogInputIO[E_aAnalogInputIO_Index.E_PV_Exhaust_Pressure]),Output=>JhValue_EXHAUST);
END_ACTION

END_PROGRAM

// ---- POUs/P92_Maintenance.TcPOU
PROGRAM P92_Maintenance
VAR
	(* Input *)
	//Light
	rTrigReactorCabinetSwitch	: R_TRIG;
	rTrigReactorCabinetMagnet 	: R_TRIG;
	fTrigReactorCabinetMagnet 	: F_TRIG;
	rTrigGasCabinetSwitch		: R_TRIG;
	rTrigGasCabinetMagnet		: R_TRIG;
	fTrigGasCabinetMagnet		: F_TRIG;

	bReactorCabinetLampSwitch : BOOL;
	bGasCabinetLampSwitch	: BOOL;
	
	bReactorCabientMagnet	: BOOL;
	bGasCabinetMagnet		: BOOL;
	bPowerDistributeMagnet	: BOOL;
	
	(* Output to Device *)
	// Cabinet Lamp
	bReactorCabinetLamp		: BOOL;
	bGasCabinetLamp			: BOOL;
	bPowerDistributeLamp	: BOOL;
	
	bSMPS24V480WFault		: BOOL;
	bSMPS24V72WFault		: BOOL;
	bSMPS15VPlusFault		: BOOL;
	bSMPS15VMinusFault		: BOOL;
	// Signal Tower
	bSignalTower			: BYTE;
	TimerSignalTower		: TON;
	bBuzzer					: BOOL;
END_VAR

(* Read from Device Value *)

// Reactor Cabinet Lamp
rTrigReactorCabinetSwitch(CLK:=GVL_IO_REACTOR_CABINET.DI_01_ReactorCabinetLampButton);
fTrigReactorCabinetMagnet(CLK:=GVL_IO_REACTOR_CABINET.DI_03_ReactorCabinetDoorClose);

IF rTrigReactorCabinetSwitch.Q OR rTrigReactorCabinetMagnet.Q OR fTrigReactorCabinetMagnet.Q THEN
	bReactorCabinetLamp := NOT(bReactorCabinetLamp);
END_IF
// Gas Delivery Cabinet Lamp
rTrigGasCabinetSwitch(CLK:= GVL_IO_GAS_CABINET.DI_01_GasCabinetLampButton);
rTrigGasCabinetMagnet(CLK:= GVL_IO_GAS_CABINET.DI_01_GasCabinetDoorClose);

IF rTrigGasCabinetSwitch.Q THEN
	bGasCabinetLamp := NOT(bGasCabinetLamp);
ELSIF fTrigGasCabinetMagnet.Q THEN
	bGasCabinetLamp := TRUE;
ELSIF rTrigGasCabinetMagnet.Q THEN
	bGasCabinetLamp := FALSE;
END_IF

IF GVL_IO_GAS_CABINET.DI_01_ControlCabinetDoorClose = TRUE THEN
	IF bPowerDistributeLamp THEN 
		bPowerDistributeLamp:=FALSE;
	END_IF
ELSE
	bPowerDistributeLamp := NOT(bPowerDistributeMagnet); //Magnet Switch	
END_IF
// Power Distribute Unit Lamp


_Action_Buzzer();
_Action_SignalTower();

(* Write to Device Value *)
GVL_IO_REACTOR_CABINET.DO_06_ReactorCabinetLamp := bReactorCabinetLamp;
GVL_IO_GAS_CABINET.DO_07_GasCabinetLamp := bGasCabinetLamp;
GVL_IO_GAS_CABINET.DO_07_ControlCabinetLamp := bPowerDistributeLamp;

ACTION _Action_Buzzer:
(* Buzzer On/Off *)
IF bBuzzer <> GVL_IO.aInterlockEnable[1].2 THEN
	bBuzzer := GVL_IO.aInterlockEnable[1].2;
END_IF
END_ACTION

ACTION _Action_SignalTower:

(* Blink Signal Tower *)
CASE GVL_IO.nCaseSignalTower OF
	1: //RED 
		TimerSignalTower(IN:=TRUE, PT:=T#500MS);
		IF TimerSignalTower.Q THEN
			TimerSignalTower(IN:=FALSE);
			IF bSignalTower = 0 THEN
				bSignalTower := 2#0000_0001; // RED
			ELSE
				bSignalTower := 0;
			END_IF
		END_IF

	2: //YELLOW 
		TimerSignalTower(IN:=TRUE, PT:=T#1S);
		IF TimerSignalTower.Q THEN
			TimerSignalTower(IN:=FALSE);
			IF bSignalTower = 0 THEN
				bSignalTower := 2#0000_0010; // YELLOW
			ELSE
				bSignalTower := 0;
			END_IF
		END_IF
	3: //GREEN
		TimerSignalTower(IN:=TRUE, PT:=T#1S);
		IF TimerSignalTower.Q THEN
			TimerSignalTower(IN:=FALSE);
			IF bSignalTower = 0 THEN
				bSignalTower := 2#0000_0100; // GREEN
			ELSE
				bSignalTower := 0;
			END_IF
		END_IF
	4: //BLUE
		bSignalTower := 2#0000_1000;
	5: //WHITE
		bSignalTower := 2#0001_0000;
END_CASE

GVL_IO_REACTOR_CABINET.DO_04_SignalTowerRed:=bSignalTower.0; //0:RED-Alarm,
GVL_IO_REACTOR_CABINET.DO_04_SignalTowerOrange:=bSignalTower.1; //1:YELLOW,-Warning
GVL_IO_REACTOR_CABINET.DO_04_SignalTowerGreen:=bSignalTower.2; //2:GREEN-Running
GVL_IO_REACTOR_CABINET.DO_04_SignalTowerBlue:=bSignalTower.3; //3:BLUE-Idle
GVL_IO_REACTOR_CABINET.DO_04_SignalTowerWhite:=bSignalTower.4; //4:WHITE-Maint
GVL_IO_REACTOR_CABINET.DO_04_SignalTowerBuzzer:=bBuzzer; //5:BUZZER-Alarm
END_ACTION

END_PROGRAM
